TYPE "ATEQRecipe"
VERSION : 0.1
   STRUCT
      RessureCurrentValueUL : Real;
      RessureCurrentValueLL : Real;
      LeakCurrentValueUL : Real;
      LeakCurrentValueLL : Real;
      PositivePressureProgNo : Int;
      NegativePressureProgNo : Int;
   END_STRUCT;

END_TYPE

